{attribute 'linkalways'} 
{attribute 'no_explicit_call' := 'This FB is a CLASS and must be accessed using methods or properties'}
{attribute 'enable_dynamic_creation'}
FUNCTION_BLOCK FINAL OR_LINT EXTENDS Node
VAR
	in1 : _LINT(0);
	in2 : _LINT(0);
	out : _LINT(0);
END_VAR

METHOD PUBLIC Clone : I_Node
VAR
	pNode : POINTER TO OR_LINT;
END_VAR
pNode := __NEW(OR_LINT);
Clone := pNode^;
END_METHOD

METHOD FB_init : BOOL
VAR_INPUT
	bInitRetains : BOOL; // if TRUE, the retain variables are initialized (warm start / cold start)
	bInCopyCode : BOOL;  // if TRUE, the instance afterwards gets moved into the copy code (online change)
END_VAR
AddInput('in1',THIS^.in1);
AddInput('in2',THIS^.in2);
AddOutput('out', THIS^.out);
END_METHOD

METHOD PROTECTED OnExecute
VAR
END_VAR
out.Value := in1.Value OR in2.Value;
END_METHOD

END_FUNCTION_BLOCK

(* stored: Version 1.1.0.1, ProductVersion 3.1.4024.15
   POU OR_LINT: Id {903b0d21-ddd4-416f-849a-f8ca4b3c3c4c}, SpecialFunc None
   Folder Constructor: Id {3d11be2c-6f8e-431e-a6c4-ec23192fef6f}
   Method Clone: Id {5cdc7b31-3847-45cd-85f1-f4acd923da30}
   Method FB_init: Id {47358c2c-ba65-48c4-bad3-4655c9452984}
   Method OnExecute: Id {17d4022a-ba84-481d-b7ad-7014facb7640} *)
